TEXTLIST CoordSystem
  0 = 'ACS'
  1 = 'MCS'
  2 = 'WCS'
  3 = 'PCS_1'
  4 = 'PCS_2'
  5 = 'TCS'
  6 = 'ICS'
   = ''
END_TEXTLIST

(* stored: Version 1.1.0.1
   TextList CoordSystem: Id {cbd89d38-a861-4ab9-a941-7e234ed51a0d} *)
